// TIA Portal project "Demo_Project" (V17)

(* hardware
DEVICE "PLC_1"  S7-1200 Station
   slot 0: "Rack_0"  S7-1200 Rack  Rack  V1.0
   slot 1: "PLC_1"  CPU 1214C DC/DC/DC  6ES7 214-1AG40-0XB0  V4.5
*)

// ===== PLC "PLC_1"  CPU 1214C DC/DC/DC =====

VAR_GLOBAL   // PLC tag table "IO_Tags"
   "Start_Button" AT %I0.0 : Bool;
   "Stop_Button" AT %I0.1 : Bool;
   "Motor_Run" AT %Q0.0 : Bool;
   "Motor_Fault" AT %I0.2 : Bool;
END_VAR

DATA_BLOCK "DB_Motor"   // DB1
{ S7_Optimized_Access := 'TRUE' }
VERSION : 0.1
   VAR
      Motor_Status : Bool := FALSE;   // 电机运行状态
      Start_Latch : Bool := FALSE;   // 启动自锁
      Run_Hours : Real := 0.0;   // 运行小时数
   END_VAR
BEGIN
END_DATA_BLOCK

FUNCTION "Motor_Control" : Void   // FC1, LAD
{ S7_Optimized_Access := 'TRUE' }
VERSION : 0.1
BEGIN

REGION Network 1: 启动自锁
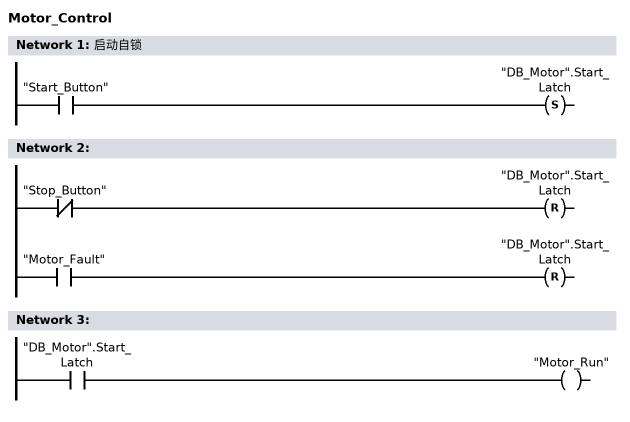
   RUNG wire#powerrail
      Contact( "Start_Button" )
      S_Coil( "DB_Motor".Start_Latch )
   END_RUNG
   // the same network as SCL:
   IF "Start_Button" THEN "DB_Motor".Start_Latch := TRUE; END_IF;
END_REGION

REGION Network 2
   RUNG wire#powerrail
      I_Contact( "Stop_Button" )
      R_Coil( "DB_Motor".Start_Latch )
   END_RUNG
   RUNG wire#powerrail
      Contact( "Motor_Fault" )
      R_Coil( "DB_Motor".Start_Latch )
   END_RUNG
   // the same network as SCL:
   IF NOT "Stop_Button" THEN "DB_Motor".Start_Latch := FALSE; END_IF;
   IF "Motor_Fault" THEN "DB_Motor".Start_Latch := FALSE; END_IF;
END_REGION

REGION Network 3
   RUNG wire#powerrail
      Contact( "DB_Motor".Start_Latch )
      Coil( "Motor_Run" )
   END_RUNG
   // the same network as SCL:
   "Motor_Run" := "DB_Motor".Start_Latch;
END_REGION
END_FUNCTION

ORGANIZATION_BLOCK "Main"   // OB1, LAD, ProgramCycle
TITLE = "Main Program Sweep (Cycle)"
{ S7_Optimized_Access := 'TRUE' }
VERSION : 0.1
   VAR_INPUT
      Initial_Call : Bool;   // Initial call of this OB
      Remanence : Bool;   // =True, if remanent data are available
   END_VAR
BEGIN
END_ORGANIZATION_BLOCK